PROGRAM Flasher
VAR
	Timer2: BOOL;
	Timer1: BOOL;
	FlashingLight: BOOL;
	Timer1TON: TON;
	Timer2TON: TON;
	FlashingLight2: BOOL;
	Timer3TON: TON;
	TonToInt: INT;
	LessThanTimer: BOOL;
	Result: UINT;
	SomeOut: BOOL;
	Ton3Elapsed: TIME;
	Timer3: BOOL;
END_VAR

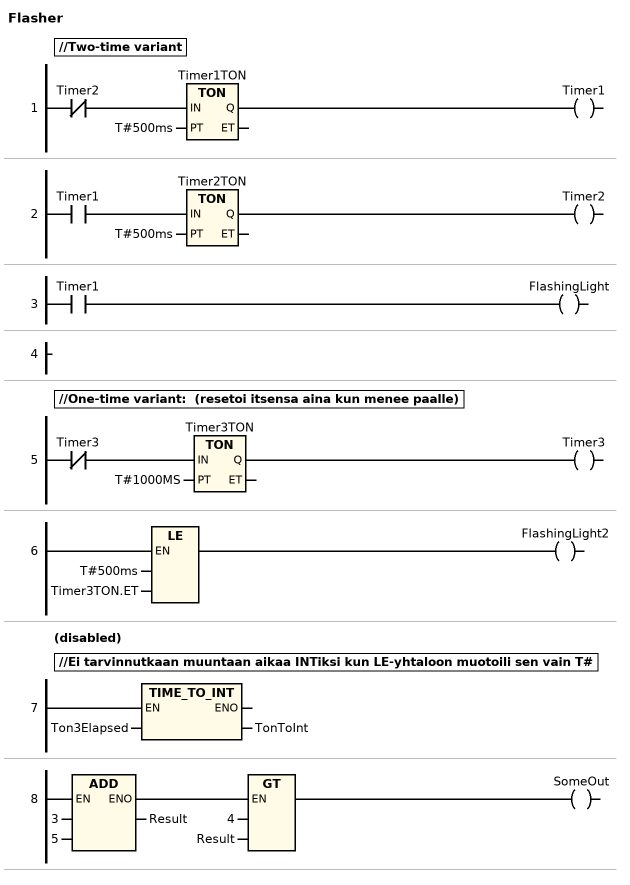
// NETWORK 1
// label: //Two-time variant
Timer1TON(IN := NOT Timer2, PT := T#500ms); // TON
Timer1 := Timer1TON.Q;

// NETWORK 2
Timer2TON(IN := Timer1, PT := T#500ms); // TON
Timer2 := Timer2TON.Q;

// NETWORK 3
FlashingLight := Timer1;

// NETWORK 4

// NETWORK 5
// label: //One-time variant:  (resetoi itsensa aina kun menee paalle)
Timer3TON(IN := NOT Timer3, PT := T#1000MS); // TON
Timer3 := Timer3TON.Q;

// NETWORK 6
FlashingLight2 := T#500ms <= Timer3TON.ET;

// NETWORK 7 (disabled)
// label: //Ei tarvinnutkaan muuntaan aikaa INTiksi kun LE-yhtaloon muotoili sen vain T#
// TonToInt := TIME_TO_INT(Ton3Elapsed);

// NETWORK 8
Result := 3 + 5;
SomeOut := 4 > Result;

END_PROGRAM

(* stored: Version 1.1.0.1, ProductVersion 3.1.4024.10
   POU Flasher: Id {1951a133-f9df-4b0e-bb9e-a1679fe79f1f}, SpecialFunc None *)
